//{attribute 'qualified_only'}
{attribute 'strict'}
TYPE eAndMethod :
(
	Minimum,
	Product
);
END_TYPE

(* stored: Version 1.1.0.1, ProductVersion 3.1.4024.6
   DUT eAndMethod: Id {8f6c04f7-111d-4201-b0b9-b63752785150} *)
